IO5:  NOP   0;
      NOP   0;
// --- FCM 06 - Fresh air flap ---
      L     "MAL1S023Par".Ilo.ILOMode;
      L     6;
      <>I   ;
      SPB   IO6;
// man on
      U     "MAL1S023Par".Ilo.GrCMDManOn[1];
      S     "G231M".Gr.InManual; // FRESH AIR LOUVER  GERM 7
//      R     DB909.DBX 3032.0
// man off
      U     "MAL1S023Par".Ilo.GrCMDManOff[1];
      S     "G231M".Gr.CmdManualOff; // FRESH AIR LOUVER  GERM 7
      R     "G231M".Gr.InManual; // FRESH AIR LOUVER  GERM 7
      R     "G231M".USW14; // ILO-cmd
      R     "G231M".USW15; // ILO-cmd
      R     "MAL1S023Par".Ilo.GrCMDManOff[1];
      R     "MAL1S023Par".Ilo.GrCMDManAdditional.Cmd1[1];
      R     "MAL1S023Par".Ilo.GrCMDManAdditional.Cmd2[1];
// man start
      U     "MAL1S023Par".Ilo.GrCMDManStart[1];
      S     "G231M".Gr.CmdOn; // FRESH AIR LOUVER  GERM 7
      S     "G231M".Gr.CmdContinue; // FRESH AIR LOUVER  GERM 7
      R     "MAL1S023Par".Ilo.GrCMDManStart[1];
      U     "MAL1S023Par".Ilo.GrCMDManStart[2];
      R     "MAL1S023Par".Ilo.GrCMDManStart[2];

      U     "MAL1S023Par".Ilo.GrCMDManOn[1];
      R     "MAL1S023Par".Ilo.GrCMDManOn[1];
// man stop
      U     "MAL1S023Par".Ilo.GrCMDManStop[1];
      S     "G231M".Gr.CmdOff; // FRESH AIR LOUVER  GERM 7
      R     "MAL1S023Par".Ilo.GrCMDManStop[1];
// man fault reset
//BRT070310      U     "MAL1S023Par".Ilo.GrCMDManOn[17]
      U     "MAL1S023Par".Ilo.GrCMDManFaultReset[1]; //BRT070310
      S     "G231M".Gr.CmdFaultReset; // FRESH AIR LOUVER  GERM 7
//MW  R     "MAL1S023Par".Ilo.GrCMDManOn[17]
      R     "MAL1S023Par".Ilo.GrCMDManFaultReset[1];
// moving direction

// target position
      UN    "G231M".Gr.InManual; // FRESH AIR LOUVER  GERM 7
      SPB   F06b;
      L     "MAL1S023Par".Ilo.SetpointInt01[1];
      T     "MAL1S023Par".Par.ParIntProcess.TarPos_ILO_FreshAir;
F06b: NOP   0;

IO6:  NOP   0;
      NOP   0;
// --- FCM 09 - Floor drives ---
      L     "MAL1S023Par".Ilo.ILOMode;
      L     9;
      <>I   ;
      SPB   IO9;
// man on
      U     "MAL1S023Par".Ilo.GrCMDManOn[1];
      S     "G013G".Gr.InManual; // GENERAL ELEMENTS GERM 7
      S     "G225M".Gr.InManual; // TRAVELLING DRIVE  GERM 7
      S     "G229M".Gr.InManual; // TURNING SCREWS  GERM 7
      R     "MAL1S023Par".Ilo.GrCMDManOn[1];
// man off
      U     "MAL1S023Par".Ilo.GrCMDManOff[1];
      S     "G013G".Gr.CmdManualOff; // GENERAL ELEMENTS GERM 7
      R     "G013G".Gr.InManual; // GENERAL ELEMENTS GERM 7
      S     "G225M".Gr.CmdManualOff; // TRAVELLING DRIVE  GERM 7
      R     "G225M".Gr.InManual; // TRAVELLING DRIVE  GERM 7
      R     "G225M".USW14; // ILO-cmd
      R     "G225M".USW15; // ILO-cmd
      S     "G229M".Gr.CmdManualOff; // TURNING SCREWS  GERM 7
      R     "G229M".Gr.InManual; // TURNING SCREWS  GERM 7
      R     "G229M".USW14; // ILO-cmd
      R     "G229M".USW15; // ILO-cmd
      R     "MAL1S023Par".Ilo.GrCMDManOff[1];
      R     "MAL1S023Par".Ilo.GrCMDManAdditional.Cmd1[1];
      R     "MAL1S023Par".Ilo.GrCMDManAdditional.Cmd2[1];
// man start
      U     "MAL1S023Par".Ilo.GrCMDManStart[1];
      S     "G013G".Gr.CmdOn; // GENERAL ELEMENTS GERM 7
      S     "G013G".Gr.CmdContinue; // GENERAL ELEMENTS GERM 7
      S     "G225M".Gr.CmdOn; // TRAVELLING DRIVE  GERM 7
      S     "G225M".Gr.CmdContinue; // TRAVELLING DRIVE  GERM 7
      S     "G229M".Gr.CmdOn; // TURNING SCREWS  GERM 7
      S     "G229M".Gr.CmdContinue; // TURNING SCREWS  GERM 7
      U     "MAL1S023Par".Ilo.GrCMDManStart[1];
      R     "MAL1S023Par".Ilo.GrCMDManStart[1];
      U     "MAL1S023Par".Ilo.GrCMDManStart[2];
      R     "MAL1S023Par".Ilo.GrCMDManStart[2];
// man stop
      U     "MAL1S023Par".Ilo.GrCMDManStop[1];
//====>BRT070310 - vom Man Off rauskopiert nach Man Stop
      O(    ;
      U(    ;
      U     "G225M".A_2711_BZS46.StTrue; // stop discharge side
      O     "G225M".A_2711_BZS46.InpTrue;
      U     "G225M".Gr.InManual;
      U     "G225M".USW14; // ILO-cmd run fwd
      )     ;
      O(    ;
      U     "G225M".A_2711_BZS44.StTrue; // stop fan side
      O     "G225M".A_2711_BZS44.InpTrue; // stop fan side
      U     "G225M".Gr.InManual;
      U     "G225M".USW15; // ILO-cmd run rev
      )     ;
      U(    ;
      L     "MAL1S023Par".Ilo.ILOMode;
//BRT070310      L     8
      L     9; //BRT070310
      ==I   ;
      )     ;
      )     ;
//<====BRT070310
      S     "G225M".Gr.CmdOff; // TRAVELLING DRIVE  GERM 7
//BRT120310      S     "G229M".Gr.CmdOff           // TURNING SCREWS  GERM 7
      R     "G225M".USW14; // ILO-cmd run fwd  //BRT120310
      R     "G225M".USW15; // ILO-cmd run rev  //BRT120310
      R     "MAL1S023Par".Ilo.GrCMDManStop[1];
// man fault reset
      U     "MAL1S023Par".Ilo.GrCMDManFaultReset[1];
      S     "G013G".Gr.CmdFaultReset; // GENERAL ELEMENTS GERM 7
      S     "G225M".Gr.CmdFaultReset; // TRAVELLING DRIVE  GERM 7
      S     "G229M".Gr.CmdFaultReset; // TURNING SCREWS  GERM 7
      R     "MAL1S023Par".Ilo.GrCMDManFaultReset[1];
// manual direction
      UN    "G225M".Gr.InManual; // TRAVELLING DRIVE  GERM 7
      SPB   f092;
      U     "MAL1S023Par".Ilo.GrCMDManAdditional.Cmd1[1];
      =     "G225M".USW14; // ILO-cmd run fwd
      U     "MAL1S023Par".Ilo.GrCMDManAdditional.Cmd2[1];
      =     "G225M".USW15; // ILO-cmd run rev
// target position
      L     "MAL1S023Par".Ilo.SetpointInt01[1];
      T     "MAL1S023Par".Par.ParIntProcess.Speed_ILO_FloorRotating;
f092: NOP   0;


IO9:  NOP   0;
// --- FCM 10 - local operating on operating panels ---

      L     "MAL1S023Par".Ilo.ILOMode;
      L     10;
      <>I   ;
      SPB   I10;
// man on
      U     "MAL1S023Par".Ilo.GrCMDManOn[1];
      S     "G013G".Gr.InManual; // GENERAL ELEMENTS GERM 7
      S     "G225M".Gr.InManual; // Traveling  Drive Germatingbox 7
      S     "G229M".Gr.InManual; // Turning Screws Germinationbox 7
      S     "G224M".Gr.InManual; // Wall locking Germatingbox 7
      S     "G222M".Gr.InManual; // Backwall moving Germatingbox 7
      S     "G223M".Gr.InManual; // Discharger locking Germatingbox 7
      R     "MAL1S023Par".Ilo.GrCMDManOn[1];
// man off
      U     "MAL1S023Par".Ilo.GrCMDManOff[1];
      S     "G013G".Gr.CmdManualOff; // GENERAL ELEMENTS GERM 7
      R     "G013G".Gr.InManual; // GENERAL ELEMENTS GERM 7
      S     "G225M".Gr.CmdManualOff; // Traveling  Drive Germatingbox 7
      R     "G225M".Gr.InManual; // Traveling  Drive Germatingbox 7
      R     "G225M".USW14; // ILO-cmd
      R     "G225M".USW15; // ILO-cmd
      S     "G229M".Gr.CmdManualOff; // Turning Screws Germinationbox 7
      R     "G229M".Gr.InManual; // Turning Screws Germinationbox 7
      R     "G229M".USW14; // ILO-cmd
      R     "G229M".USW15; // ILO-cmd
      S     "G224M".Gr.CmdManualOff; // Wall locking Germatingbox 7
      R     "G224M".Gr.InManual; // Wall locking Germatingbox 7
      S     "G223M".Gr.CmdManualOff; // Discharger locking Germatingbox 7
      R     "G223M".Gr.InManual; // Discharger locking Germatingbox 7
      S     "G222M".Gr.CmdManualOff; // Backwall moving Germatingbox 7
      R     "G222M".Gr.InManual; // Backwall moving Germatingbox 7
      R     "MAL1S023Par".Ilo.GrCMDManOff[1];
      R     "MAL1S023Par".Ilo.GrCMDManAdditional.Cmd1[1];
      R     "MAL1S023Par".Ilo.GrCMDManAdditional.Cmd2[1];
// man start
      U     "G227M".A_2711_KCL01I1.InpTrue; // pushbutton "start screws"
      S     "G013G".Gr.CmdOn; // GENERAL ELEMENTS GERM 7
      S     "G013G".Gr.CmdContinue; // GENERAL ELEMENTS GERM 7
      S     "G229M".Gr.CmdOn; // Turning Screws Germinationbox 7
      S     "G229M".Gr.CmdContinue; // Turning Screws Germinationbox 7
      S     "G225M".Gr.CmdOn; // Traveling  Drive Germatingbox 7
      S     "G225M".Gr.CmdContinue; // Traveling  Drive Germatingbox 7
      U     "MAL1S023Par".Ilo.GrCMDManStart[1];
      R     "MAL1S023Par".Ilo.GrCMDManStart[1];
      U     "MAL1S023Par".Ilo.GrCMDManStart[2];
      R     "MAL1S023Par".Ilo.GrCMDManStart[2];
// man stop
      UN    "G227M".A_2711_KCL01I2.InpTrue; // pushbutton "stop screws"  //dyk 081025 Inverted
      S     "G229M".Gr.CmdOff; // Turning Screws Germinationbox 7
      U     "MAL1S023Par".Ilo.GrCMDManStop[1];
      O(    ;
      UN    "G227M".A_2711_KCL01I3.InpTrue; // pushbutton "drive fwd"
      UN    "G227M".A_2711_KCL01I4.InpTrue; // pushbutton "drive rev"
      )     ;
      S     "G225M".Gr.CmdOff; // Traveling  Drive Germatingbox 7

      UN    "G224M".Gr.InManual; // Wall locking Germatingbox 7
      O(    ;
      UN    "G227M".A_2715_KCL01I5.InpTrue; // pushbutton "locking"
      UN    "G227M".A_2715_KCL01I6.InpTrue; // pushbutton "unlocking"
      )     ;
      S     "G224M".Gr.CmdOff; // Wall locking/unlocking Germatingbox 7

      UN    "G223M".Gr.InManual; // discharger coupling Germatingbox 7
      O(    ;
      UN    "G227M".A_2715_KCL01I4.InpTrue; // pushbutton "discharger coupling"
      UN    "G227M".A_2715_KCL01I3.InpTrue; // pushbutton "discharger uncoupling"
      )     ;
      S     "G223M".Gr.CmdOff; // discharger coupling Germatingbox 7

      UN    "G222M".Gr.InManual; // Backwall moving Germatingbox 7
      O(    ;
      UN    "G227M".A_2715_KCL01I1.InpTrue; // pushbutton "backwall lifting"
      UN    "G227M".A_2715_KCL01I2.InpTrue; // pushbutton "backwall lowerring"
      )     ;
      S     "G222M".Gr.CmdOff; // Backwall moving Germatingbox 7

      U     "MAL1S023Par".Ilo.GrCMDManStop[1];
      R     "MAL1S023Par".Ilo.GrCMDManStop[1];
// man fault reset
      U     "MAL1S023Par".Ilo.GrCMDManFaultReset[1];
      S     "G013G".Gr.CmdFaultReset; // GENERAL ELEMENTS GERM 7
      S     "G225M".Gr.CmdFaultReset; // Traveling  Drive Germatingbox 7
      S     "G229M".Gr.CmdFaultReset; // Turning Screws Germinationbox 7
      R     "MAL1S023Par".Ilo.GrCMDManFaultReset[1];
      NOP   0;
// Manual wall locking
      UN    "G224M".Gr.InManual; // Wall locking Germatingbox 7
      ON    "G227M".A_2715_KCL01I5.InpTrue; // pushbutton "locking"
      SPB   f102;
      S     "G224M".Gr.CmdOn; // Wall locking/unlocking Germatingbox 7
f102: NOP   0;
// Manual wall unlocking
      UN    "G224M".Gr.InManual; // Wall locking Germatingbox 7
      ON    "G227M".A_2715_KCL01I6.InpTrue; // pushbutton "unlocking"
      SPB   f103;
      S     "G224M".Gr.CmdOn; // Wall locking/unlocking Germatingbox 7
f103: NOP   0;
// Manual discharger coupling
      UN    "G223M".Gr.InManual; // discharger coupling Germatingbox 7
      ON    "G227M".A_2715_KCL01I4.InpTrue; // pushbutton "discharger coupling"
      SPB   f104;
      S     "G223M".Gr.CmdOn; // discharger coupling Germatingbox 7
f104: NOP   0;
// Manual discharger uncoupling
      UN    "G223M".Gr.InManual; // discharger coupling Germatingbox 7
      ON    "G227M".A_2715_KCL01I3.InpTrue; // pushbutton "discharger uncoupling"
      SPB   f105;
      S     "G223M".Gr.CmdOn; // discharger coupling Germatingbox 7
f105: NOP   0;
// Manual backwall moving
      UN    "G222M".Gr.InManual; // Backwall moving Germatingbox 7
      ON    "G227M".A_2715_KCL01I1.InpTrue; // pushbutton "backwall lifting"
      SPB   f106;
      S     "G222M".Gr.CmdOn; // Backwall moving Germatingbox 7
f106: NOP   0;
      UN    "G222M".Gr.InManual; // Backwall moving Germatingbox 7
      ON    "G227M".A_2715_KCL01I2.InpTrue; // pushbutton "backwall lowerring"
      SPB   f107;
      S     "G222M".Gr.CmdOn; // Backwall moving Germatingbox 7
f107: NOP   0;
// manual direction
      UN    "G225M".Gr.InManual; // Traveling  Drive Germatingbox 7
      O     ;
      UN    "G227M".A_2711_KCL01I3.InpTrue; // pushbutton "drive fwd"
      UN    "G227M".A_2711_KCL01I4.InpTrue; // pushbutton "drive rev"
      SPB   f109;
      U     "G227M".A_2711_KCL01I3.InpTrue; // pushbutton "drive fwd"
      =     "G225M".USW14; // ILO-cmd run fwd
      S     "G225M".Gr.CmdOn; // Traveling  Drive Germatingbox 7
      U     "G227M".A_2711_KCL01I4.InpTrue; // pushbutton "drive rev"
      =     "G225M".USW15; // ILO-cmd run rev
      S     "G225M".Gr.CmdOn; // Traveling  Drive Germatingbox 7

// target position
      L     "MAL1S023Par".Ilo.SetpointInt01[1];
      T     "MAL1S023Par".Par.ParIntProcess.Speed_ILO_FloorRotating;
f109: NOP   0;

I10:  NOP   0;
//
// copy state
      U     "G225M".Gr.InOutAutostartMan; // TRAVELLING DRIVE  GERM 7
      =     "MAL1S023Par".Ilo.GrSTMan[2];
      U     "G229M".Gr.InOutAutostartMan; // TURNING SCREWS  GERM 7
      =     "MAL1S023Par".Ilo.GrSTMan[6];
      U     "G230M".Gr.InOutAutostartMan; // FAN AND VALVE SRAY AIR  GERM 7
      =     "MAL1S023Par".Ilo.GrSTMan[7];
      U     "G231M".Gr.InOutAutostartMan; // FRESH AIR LOUVER  GERM 7
      =     "MAL1S023Par".Ilo.GrSTMan[8];
      U     "G237M".Gr.InOutAutostartMan; // COOLING / HEATING  GERM 7
      =     "MAL1S023Par".Ilo.GrSTMan[14];

// copy state

NETWORK
TITLE =ASW_9999: Init ASW Flags
// clear all flags explicde to find them back
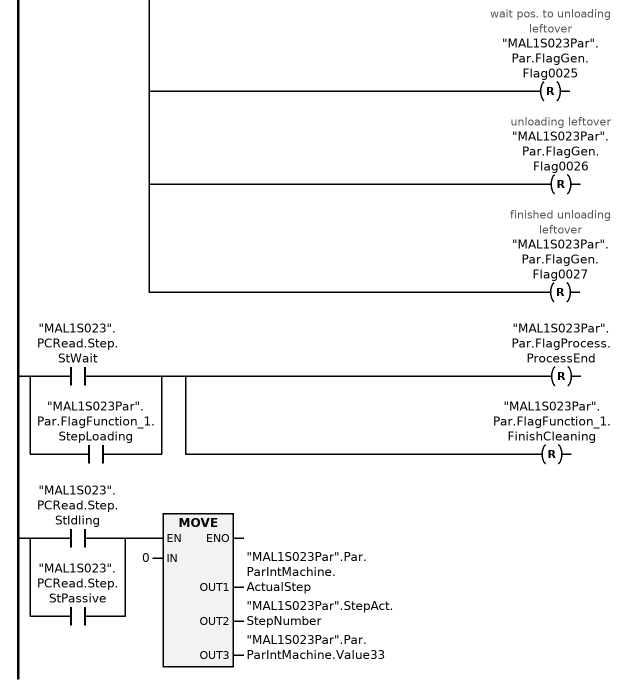
      U     "MAL1S023".PCRead.Step.StIdling;
      O     "MAL1S023".PCRead.Step.StPassive;
      R     "MAL1S023Par".Par.FlagFunction_1.StepLoading;
      R     "MAL1S023Par".Par.FlagFunction_1.StepUnloading;
      R     "MAL1S023Par".Par.FlagFunction_1.StepCleaning;
      R     "MAL1S023Par".Par.FlagFunction_1.LoadingBreak;
      R     "MAL1S023Par".Par.FlagFunction_1.UnloadingBreak;
      R     "MAL1S023Par".Par.FlagFunction_1.CleaningBreak;
      R     "MAL1S023Par".Par.FlagFunction_1.FinishLoading;
      R     "MAL1S023Par".Par.FlagFunction_1.FinishUnloading;
      R     "MAL1S023Par".Par.FlagFunction_1.FinishCleaning;
      R     "MAL1S023Par".Par.FlagFunction_1.Round_1;
      R     "MAL1S023Par".Par.FlagFunction_1.Round_2;
      R     "MAL1S023Par".Par.FlagFunction_1.Round_3;
      R     "MAL1S023Par".Par.FlagFunction_1.Round_4;
      R     "MAL1S023Par".Par.FlagFunction_1.Round_5;
      R     "MAL1S023Par".Par.FlagFunction_1.Round_6;
      R     "MAL1S023Par".Par.FlagFunction_1.Beladung_beendet;
      R     "MAL1S023Par".Par.FlagFunction_1.Entladerunden_erreicht;
      R     "MAL1S023Par".Par.FlagFunction_1.Reinigungsrunde_erreicht;
      R     "MAL1S023Par".Par.FlagGen.TurningStarted;
      R     "MAL1S023Par".Par.FlagFunction_1.TurningStart;
      R     "MAL1S023Par".Par.FlagFunction_1.TurningStop;
      R     "MAL1S023Par".Par.FlagFunction_1.TurningLeft;
      R     "MAL1S023Par".Par.FlagFunction_1.TurningRight;
      R     "MAL1S023Par".Par.FlagFunction_1.LoadFirstPartEnd;
      R     "MAL1S023Par".Par.FlagFunction_1.TurningWithSpraying;
      R     "MAL1S023Par".Par.FlagFunction_1.TurningWithoutSpraying;
      R     "MAL1S023Par".Par.FlagGen.TurningStarted;
      R     "MAL1S023Par".Par.FlagProcess2.Turning1WithoutSpraying;
      R     "MAL1S023Par".Par.FlagProcess2.Turning2WithoutSpraying;
      R     "MAL1S023Par".Par.FlagProcess2.Turning1WithSpraying;
      R     "MAL1S023Par".Par.FlagProcess2.Turning2WithSpraying;
      R     "MAL1S023Par".Par.FlagProcess2.Turning1WithDosing;
      R     "MAL1S023Par".Par.FlagProcess2.Turning2WithDosing;
      R     "MAL1S023Par".Par.FlagProcess2.StartFirstTurningRound;
      R     "MAL1S023Par".Par.FlagProcess2.StartSecondTurningRound;

      R     "MAL1S023Par".Par.FlagFunction_1.UnloadFirstPartEnd;
      R     "MAL1S023Par".Par.FlagFunction_1.UnloadSecondPartEnd;
      R     "MAL1S023Par".Par.FlagFunction_1.UnloadFirstPart;
      R     "MAL1S023Par".Par.FlagFunction_1.UnloadSecondPart;
      R     "MAL1S023Par".Par.FlagFunction_1.UnloadingStarted;
      R     "MAL1S023Par".Par.FlagProcess.ProcessActive;
      R     "MAL1S023Par".Par.FlagProcess.ProcessStartFP;
      R     "MAL1S023Par".Par.FlagProcess.ProcessStartScan;
      R     "MAL1S023Par".Par.FlagProcess.ProcessEnd;
      R     "MAL1S023Par".Par.FlagProcess.FP_SendResultToPIC;
      R     "MAL1S023Par".Par.FlagMachine.ImpulsNullstellung;
      R     "MAL1S023Par".Par.FlagMachine_0.CmdTurnRevAfterUnloading;
      R     "MAL1S023Par".Par.FlagMachine_0.CleaningAfterUnloading;
      R     "MAL1S023Par".Par.FlagMachine_0.CleaningAfterLoading;

      R     "MAL1S023Par".Par.FlagGen.Flag0024; // finished first unloading
      R     "MAL1S023Par".Par.FlagGen.Flag0025; // wait pos. to unloading leftover
      R     "MAL1S023Par".Par.FlagGen.Flag0026; // unloading leftover
      R     "MAL1S023Par".Par.FlagGen.Flag0027; // finished unloading leftover

//
      U     "MAL1S023".PCRead.Step.StWait;
      O     "MAL1S023Par".Par.FlagFunction_1.StepLoading;
      R     "MAL1S023Par".Par.FlagProcess.ProcessEnd;
      R     "MAL1S023Par".Par.FlagFunction_1.FinishCleaning;

      U     "MAL1S023".PCRead.Step.StIdling;
      O     "MAL1S023".PCRead.Step.StPassive;
      SPBN  csn;
      L     0; // clear step number
      T     "MAL1S023Par".Par.ParIntMachine.ActualStep;
      T     "MAL1S023Par".StepAct.StepNumber;
      T     "MAL1S023Par".Par.ParIntMachine.Value33; //aktuelle Wartezeit Maschine bei 100% Unloading-Position
csn:  NOP   0;

NETWORK
TITLE =Main0_End: Init flag
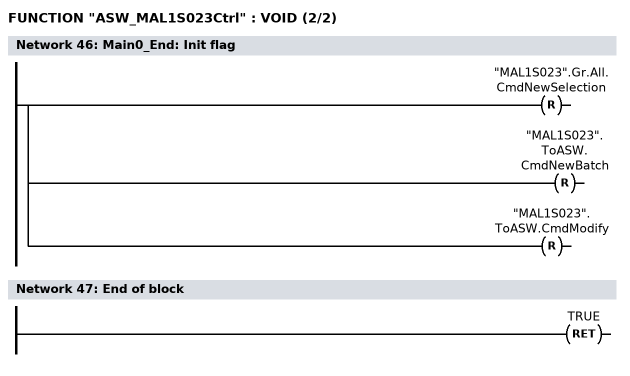

      SET   ;
      R     "MAL1S023".Gr.All.CmdNewSelection;
      R     "MAL1S023".ToASW.CmdNewBatch;
      R     "MAL1S023".ToASW.CmdModify;

NETWORK
TITLE =End of block

      BE    ;

END_FUNCTION

